// TIA Portal V20 export
VAR_GLOBAL   // PLC tag table "Default tag table"
   Clock_Byte AT %MB255 : Byte;
   Clock_10Hz AT %M255.0 : Bool;
   Clock_5Hz AT %M255.1 : Bool;
   "Clock_2.5Hz" AT %M255.2 : Bool;
   Clock_2Hz AT %M255.3 : Bool;
   "Clock_1.25Hz" AT %M255.4 : Bool;
   Clock_1Hz AT %M255.5 : Bool;
   "Clock_0.625Hz" AT %M255.6 : Bool;
   "Clock_0.5Hz" AT %M255.7 : Bool;
   System_Byte AT %MB10 : Byte;
   FirstScan AT %M10.0 : Bool;
   DiagStatusUpdate AT %M10.1 : Bool;
   AlwaysTRUE AT %M10.2 : Bool;
   AlwaysFALSE AT %M10.3 : Bool;
   mLOGIC0 AT %M0.0 : Bool;
   mAlarmDelay AT %M100.7 : Bool;
   mLOGIC1 AT %M0.1 : Bool;
   mRestart AT %M0.7 : Bool;
END_VAR
